// TIA Portal V20 export
TYPE "typeSequenceControlNodeJobInterfaceMonitoring"
// stored: Namespace Unit1.Em2
   STRUCT
      busyAutoSplice { ExternalWritable := 'False'} : Bool;
      doneAutoSplice { ExternalWritable := 'False'} : Bool;
   END_STRUCT;
END_TYPE
